% RSLogix 500 project ISO_WEEK_OF_YEAR.RSS, saved by version 9.05.01.00 %
PROJECT "ML1400"    % processor: MicroLogix 1400; MAIN_PROG %

PROGRAM FILES
  LAD 2 "MAIN_PROG"  82 rungs

DATA FILES
  O0 OUTPUT  6 elements
  I1 INPUT  8 elements
  S2 STATUS  66 elements
  B3 BINARY  53 elements
  T4 TIMER  1 elements
  C5 COUNTER  1 elements
  R6 CONTROL  1 elements
  N7 INTEGER  180 elements
  F8   1 elements

LADDER 2 "MAIN_PROG"
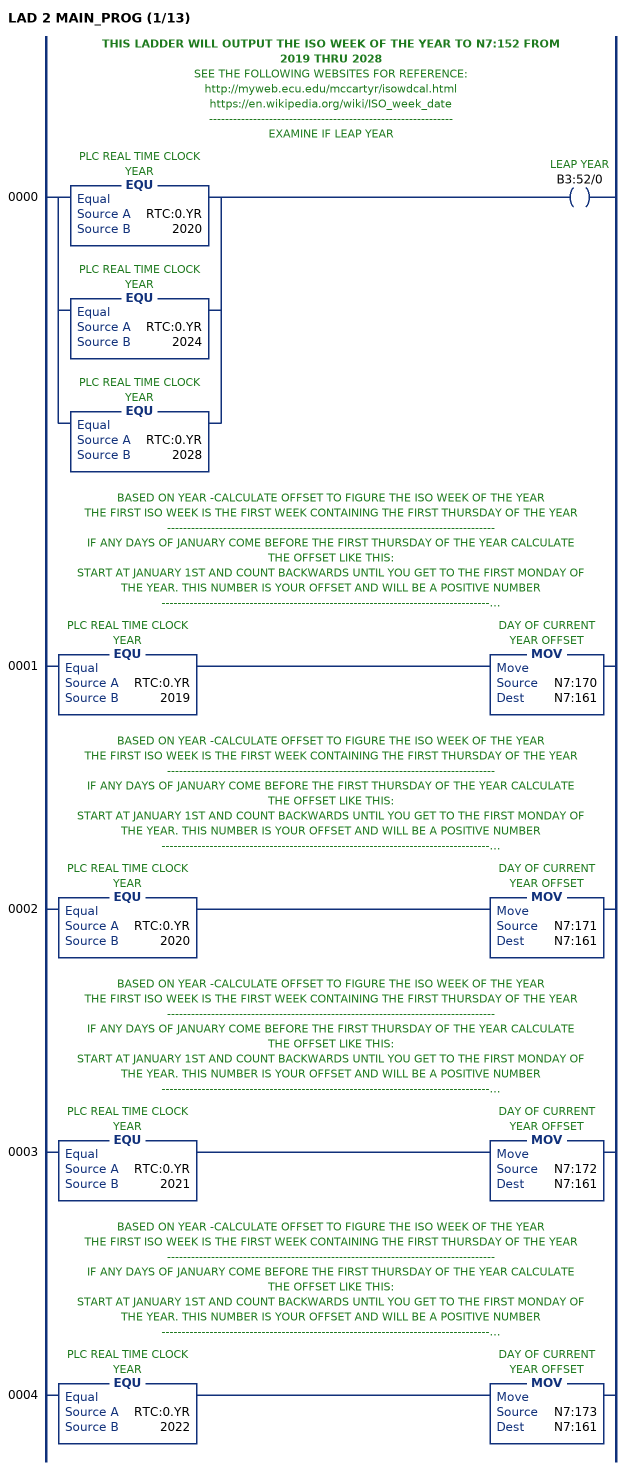
% Rung: 0 %
% TITLE: THIS LADDER WILL OUTPUT THE ISO WEEK OF THE YEAR TO N7:152 FROM 2019 THRU 2028 %
% SEE THE FOLLOWING WEBSITES FOR REFERENCE:
% http://myweb.ecu.edu/mccartyr/isowdcal.html
% https://en.wikipedia.org/wiki/ISO_week_date
% -------------------------------------------------------------
% EXAMINE IF LEAP YEAR %
SOR BST EQU RTC:0.YR 2020 NXB EQU RTC:0.YR 2024 NXB EQU RTC:0.YR 2028 BND OTE B3:52/0 EOR
%   RTC:0.YR  "PLC REAL TIME CLOCK YEAR" %
%   B3:52/0  "LEAP YEAR" %
% Rung: 1 %
% BASED ON YEAR -CALCULATE OFFSET TO FIGURE THE ISO WEEK OF THE YEAR
% THE FIRST ISO WEEK IS THE FIRST WEEK CONTAINING THE FIRST THURSDAY OF THE YEAR
% ----------------------------------------------------------------------------------
% IF ANY DAYS OF JANUARY COME BEFORE THE FIRST THURSDAY OF THE YEAR CALCULATE THE OFFSET LIKE THIS:
% START AT JANUARY 1ST AND COUNT BACKWARDS UNTIL YOU GET TO THE FIRST MONDAY OF THE YEAR. THIS NUMBER IS YOUR OFFSET AND WILL BE A POSITIVE NUMBER
% -----------------------------------------------------------------------------------
% IF NO DAYS OF JANUARY COME BEFORE THE FIRST THURSDAY OF THE YEAR CALCULATE THE OFFSET LIKE THIS:
% START AT JANUARY 1ST AND COUNT FORWARDS UNTIL YOU GET TO THE NEXT SUNDAY. THIS NUMBER IS YOUR OFFSET AND WILL BE A NEGATIVE NUMBER
% ------------------------------------------------------------------------------------
% SEE THE FOLLOWING WEBSITES FOR REFERENCE:
% http://myweb.ecu.edu/mccartyr/isowdcal.html
% https://en.wikipedia.org/wiki/ISO_week_date %
SOR EQU RTC:0.YR 2019 MOV N7:170 N7:161 EOR
%   RTC:0.YR  "PLC REAL TIME CLOCK YEAR" %
%   N7:170  "DAY OFFSET 2019" %
%   N7:161  "DAY OF CURRENT YEAR OFFSET" %
% Rung: 2 %
% BASED ON YEAR -CALCULATE OFFSET TO FIGURE THE ISO WEEK OF THE YEAR
% THE FIRST ISO WEEK IS THE FIRST WEEK CONTAINING THE FIRST THURSDAY OF THE YEAR
% ----------------------------------------------------------------------------------
% IF ANY DAYS OF JANUARY COME BEFORE THE FIRST THURSDAY OF THE YEAR CALCULATE THE OFFSET LIKE THIS:
% START AT JANUARY 1ST AND COUNT BACKWARDS UNTIL YOU GET TO THE FIRST MONDAY OF THE YEAR. THIS NUMBER IS YOUR OFFSET AND WILL BE A POSITIVE NUMBER
% -----------------------------------------------------------------------------------
% IF NO DAYS OF JANUARY COME BEFORE THE FIRST THURSDAY OF THE YEAR CALCULATE THE OFFSET LIKE THIS:
% START AT JANUARY 1ST AND COUNT FORWARDS UNTIL YOU GET TO THE NEXT SUNDAY. THIS NUMBER IS YOUR OFFSET AND WILL BE A NEGATIVE NUMBER
% ------------------------------------------------------------------------------------
% SEE THE FOLLOWING WEBSITES FOR REFERENCE:
% http://myweb.ecu.edu/mccartyr/isowdcal.html
% https://en.wikipedia.org/wiki/ISO_week_date %
SOR EQU RTC:0.YR 2020 MOV N7:171 N7:161 EOR
%   RTC:0.YR  "PLC REAL TIME CLOCK YEAR" %
%   N7:171  "DAY OFFSET 2020" %
%   N7:161  "DAY OF CURRENT YEAR OFFSET" %
% Rung: 3 %
% BASED ON YEAR -CALCULATE OFFSET TO FIGURE THE ISO WEEK OF THE YEAR
% THE FIRST ISO WEEK IS THE FIRST WEEK CONTAINING THE FIRST THURSDAY OF THE YEAR
% ----------------------------------------------------------------------------------
% IF ANY DAYS OF JANUARY COME BEFORE THE FIRST THURSDAY OF THE YEAR CALCULATE THE OFFSET LIKE THIS:
% START AT JANUARY 1ST AND COUNT BACKWARDS UNTIL YOU GET TO THE FIRST MONDAY OF THE YEAR. THIS NUMBER IS YOUR OFFSET AND WILL BE A POSITIVE NUMBER
% -----------------------------------------------------------------------------------
% IF NO DAYS OF JANUARY COME BEFORE THE FIRST THURSDAY OF THE YEAR CALCULATE THE OFFSET LIKE THIS:
% START AT JANUARY 1ST AND COUNT FORWARDS UNTIL YOU GET TO THE NEXT SUNDAY. THIS NUMBER IS YOUR OFFSET AND WILL BE A NEGATIVE NUMBER
% ------------------------------------------------------------------------------------
% SEE THE FOLLOWING WEBSITES FOR REFERENCE:
% http://myweb.ecu.edu/mccartyr/isowdcal.html
% https://en.wikipedia.org/wiki/ISO_week_date %
SOR EQU RTC:0.YR 2021 MOV N7:172 N7:161 EOR
%   RTC:0.YR  "PLC REAL TIME CLOCK YEAR" %
%   N7:172  "DAY OFFSET 2021" %
%   N7:161  "DAY OF CURRENT YEAR OFFSET" %
% Rung: 4 %
% BASED ON YEAR -CALCULATE OFFSET TO FIGURE THE ISO WEEK OF THE YEAR
% THE FIRST ISO WEEK IS THE FIRST WEEK CONTAINING THE FIRST THURSDAY OF THE YEAR
% ----------------------------------------------------------------------------------
% IF ANY DAYS OF JANUARY COME BEFORE THE FIRST THURSDAY OF THE YEAR CALCULATE THE OFFSET LIKE THIS:
% START AT JANUARY 1ST AND COUNT BACKWARDS UNTIL YOU GET TO THE FIRST MONDAY OF THE YEAR. THIS NUMBER IS YOUR OFFSET AND WILL BE A POSITIVE NUMBER
% -----------------------------------------------------------------------------------
% IF NO DAYS OF JANUARY COME BEFORE THE FIRST THURSDAY OF THE YEAR CALCULATE THE OFFSET LIKE THIS:
% START AT JANUARY 1ST AND COUNT FORWARDS UNTIL YOU GET TO THE NEXT SUNDAY. THIS NUMBER IS YOUR OFFSET AND WILL BE A NEGATIVE NUMBER
% ------------------------------------------------------------------------------------
% SEE THE FOLLOWING WEBSITES FOR REFERENCE:
% http://myweb.ecu.edu/mccartyr/isowdcal.html
% https://en.wikipedia.org/wiki/ISO_week_date %
SOR EQU RTC:0.YR 2022 MOV N7:173 N7:161 EOR
%   RTC:0.YR  "PLC REAL TIME CLOCK YEAR" %
%   N7:173  "DAY OFFSET 2022" %
%   N7:161  "DAY OF CURRENT YEAR OFFSET" %

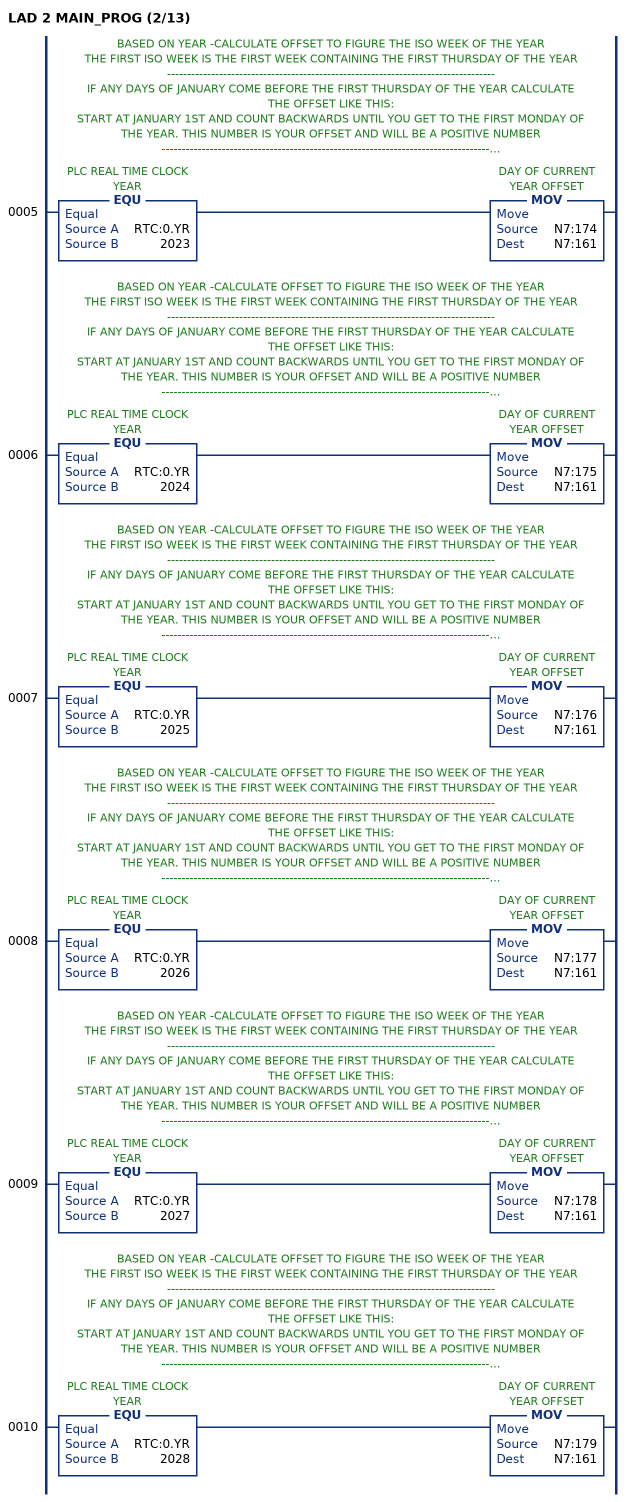
% Rung: 5 %
% BASED ON YEAR -CALCULATE OFFSET TO FIGURE THE ISO WEEK OF THE YEAR
% THE FIRST ISO WEEK IS THE FIRST WEEK CONTAINING THE FIRST THURSDAY OF THE YEAR
% ----------------------------------------------------------------------------------
% IF ANY DAYS OF JANUARY COME BEFORE THE FIRST THURSDAY OF THE YEAR CALCULATE THE OFFSET LIKE THIS:
% START AT JANUARY 1ST AND COUNT BACKWARDS UNTIL YOU GET TO THE FIRST MONDAY OF THE YEAR. THIS NUMBER IS YOUR OFFSET AND WILL BE A POSITIVE NUMBER
% -----------------------------------------------------------------------------------
% IF NO DAYS OF JANUARY COME BEFORE THE FIRST THURSDAY OF THE YEAR CALCULATE THE OFFSET LIKE THIS:
% START AT JANUARY 1ST AND COUNT FORWARDS UNTIL YOU GET TO THE NEXT SUNDAY. THIS NUMBER IS YOUR OFFSET AND WILL BE A NEGATIVE NUMBER
% ------------------------------------------------------------------------------------
% SEE THE FOLLOWING WEBSITES FOR REFERENCE:
% http://myweb.ecu.edu/mccartyr/isowdcal.html
% https://en.wikipedia.org/wiki/ISO_week_date %
SOR EQU RTC:0.YR 2023 MOV N7:174 N7:161 EOR
%   RTC:0.YR  "PLC REAL TIME CLOCK YEAR" %
%   N7:174  "DAY OFFSET 2023" %
%   N7:161  "DAY OF CURRENT YEAR OFFSET" %
% Rung: 6 %
% BASED ON YEAR -CALCULATE OFFSET TO FIGURE THE ISO WEEK OF THE YEAR
% THE FIRST ISO WEEK IS THE FIRST WEEK CONTAINING THE FIRST THURSDAY OF THE YEAR
% ----------------------------------------------------------------------------------
% IF ANY DAYS OF JANUARY COME BEFORE THE FIRST THURSDAY OF THE YEAR CALCULATE THE OFFSET LIKE THIS:
% START AT JANUARY 1ST AND COUNT BACKWARDS UNTIL YOU GET TO THE FIRST MONDAY OF THE YEAR. THIS NUMBER IS YOUR OFFSET AND WILL BE A POSITIVE NUMBER
% -----------------------------------------------------------------------------------
% IF NO DAYS OF JANUARY COME BEFORE THE FIRST THURSDAY OF THE YEAR CALCULATE THE OFFSET LIKE THIS:
% START AT JANUARY 1ST AND COUNT FORWARDS UNTIL YOU GET TO THE NEXT SUNDAY. THIS NUMBER IS YOUR OFFSET AND WILL BE A NEGATIVE NUMBER
% ------------------------------------------------------------------------------------
% SEE THE FOLLOWING WEBSITES FOR REFERENCE:
% http://myweb.ecu.edu/mccartyr/isowdcal.html
% https://en.wikipedia.org/wiki/ISO_week_date %
SOR EQU RTC:0.YR 2024 MOV N7:175 N7:161 EOR
%   RTC:0.YR  "PLC REAL TIME CLOCK YEAR" %
%   N7:175  "DAY OFFSET 2024" %
%   N7:161  "DAY OF CURRENT YEAR OFFSET" %
% Rung: 7 %
% BASED ON YEAR -CALCULATE OFFSET TO FIGURE THE ISO WEEK OF THE YEAR
% THE FIRST ISO WEEK IS THE FIRST WEEK CONTAINING THE FIRST THURSDAY OF THE YEAR
% ----------------------------------------------------------------------------------
% IF ANY DAYS OF JANUARY COME BEFORE THE FIRST THURSDAY OF THE YEAR CALCULATE THE OFFSET LIKE THIS:
% START AT JANUARY 1ST AND COUNT BACKWARDS UNTIL YOU GET TO THE FIRST MONDAY OF THE YEAR. THIS NUMBER IS YOUR OFFSET AND WILL BE A POSITIVE NUMBER
% -----------------------------------------------------------------------------------
% IF NO DAYS OF JANUARY COME BEFORE THE FIRST THURSDAY OF THE YEAR CALCULATE THE OFFSET LIKE THIS:
% START AT JANUARY 1ST AND COUNT FORWARDS UNTIL YOU GET TO THE NEXT SUNDAY. THIS NUMBER IS YOUR OFFSET AND WILL BE A NEGATIVE NUMBER
% ------------------------------------------------------------------------------------
% SEE THE FOLLOWING WEBSITES FOR REFERENCE:
% http://myweb.ecu.edu/mccartyr/isowdcal.html
% https://en.wikipedia.org/wiki/ISO_week_date %
SOR EQU RTC:0.YR 2025 MOV N7:176 N7:161 EOR
%   RTC:0.YR  "PLC REAL TIME CLOCK YEAR" %
%   N7:176  "DAY OFFSET 2025" %
%   N7:161  "DAY OF CURRENT YEAR OFFSET" %
% Rung: 8 %
% BASED ON YEAR -CALCULATE OFFSET TO FIGURE THE ISO WEEK OF THE YEAR
% THE FIRST ISO WEEK IS THE FIRST WEEK CONTAINING THE FIRST THURSDAY OF THE YEAR
% ----------------------------------------------------------------------------------
% IF ANY DAYS OF JANUARY COME BEFORE THE FIRST THURSDAY OF THE YEAR CALCULATE THE OFFSET LIKE THIS:
% START AT JANUARY 1ST AND COUNT BACKWARDS UNTIL YOU GET TO THE FIRST MONDAY OF THE YEAR. THIS NUMBER IS YOUR OFFSET AND WILL BE A POSITIVE NUMBER
% -----------------------------------------------------------------------------------
% IF NO DAYS OF JANUARY COME BEFORE THE FIRST THURSDAY OF THE YEAR CALCULATE THE OFFSET LIKE THIS:
% START AT JANUARY 1ST AND COUNT FORWARDS UNTIL YOU GET TO THE NEXT SUNDAY. THIS NUMBER IS YOUR OFFSET AND WILL BE A NEGATIVE NUMBER
% ------------------------------------------------------------------------------------
% SEE THE FOLLOWING WEBSITES FOR REFERENCE:
% http://myweb.ecu.edu/mccartyr/isowdcal.html
% https://en.wikipedia.org/wiki/ISO_week_date %
SOR EQU RTC:0.YR 2026 MOV N7:177 N7:161 EOR
%   RTC:0.YR  "PLC REAL TIME CLOCK YEAR" %
%   N7:177  "DAY OFFSET 2026" %
%   N7:161  "DAY OF CURRENT YEAR OFFSET" %
% Rung: 9 %
% BASED ON YEAR -CALCULATE OFFSET TO FIGURE THE ISO WEEK OF THE YEAR
% THE FIRST ISO WEEK IS THE FIRST WEEK CONTAINING THE FIRST THURSDAY OF THE YEAR
% ----------------------------------------------------------------------------------
% IF ANY DAYS OF JANUARY COME BEFORE THE FIRST THURSDAY OF THE YEAR CALCULATE THE OFFSET LIKE THIS:
% START AT JANUARY 1ST AND COUNT BACKWARDS UNTIL YOU GET TO THE FIRST MONDAY OF THE YEAR. THIS NUMBER IS YOUR OFFSET AND WILL BE A POSITIVE NUMBER
% -----------------------------------------------------------------------------------
% IF NO DAYS OF JANUARY COME BEFORE THE FIRST THURSDAY OF THE YEAR CALCULATE THE OFFSET LIKE THIS:
% START AT JANUARY 1ST AND COUNT FORWARDS UNTIL YOU GET TO THE NEXT SUNDAY. THIS NUMBER IS YOUR OFFSET AND WILL BE A NEGATIVE NUMBER
% ------------------------------------------------------------------------------------
% SEE THE FOLLOWING WEBSITES FOR REFERENCE:
% http://myweb.ecu.edu/mccartyr/isowdcal.html
% https://en.wikipedia.org/wiki/ISO_week_date %
SOR EQU RTC:0.YR 2027 MOV N7:178 N7:161 EOR
%   RTC:0.YR  "PLC REAL TIME CLOCK YEAR" %
%   N7:178  "DAY OFFSET 2027" %
%   N7:161  "DAY OF CURRENT YEAR OFFSET" %
% Rung: 10 %
% BASED ON YEAR -CALCULATE OFFSET TO FIGURE THE ISO WEEK OF THE YEAR
% THE FIRST ISO WEEK IS THE FIRST WEEK CONTAINING THE FIRST THURSDAY OF THE YEAR
% ----------------------------------------------------------------------------------
% IF ANY DAYS OF JANUARY COME BEFORE THE FIRST THURSDAY OF THE YEAR CALCULATE THE OFFSET LIKE THIS:
% START AT JANUARY 1ST AND COUNT BACKWARDS UNTIL YOU GET TO THE FIRST MONDAY OF THE YEAR. THIS NUMBER IS YOUR OFFSET AND WILL BE A POSITIVE NUMBER
% -----------------------------------------------------------------------------------
% IF NO DAYS OF JANUARY COME BEFORE THE FIRST THURSDAY OF THE YEAR CALCULATE THE OFFSET LIKE THIS:
% START AT JANUARY 1ST AND COUNT FORWARDS UNTIL YOU GET TO THE NEXT SUNDAY. THIS NUMBER IS YOUR OFFSET AND WILL BE A NEGATIVE NUMBER
% ------------------------------------------------------------------------------------
% SEE THE FOLLOWING WEBSITES FOR REFERENCE:
% http://myweb.ecu.edu/mccartyr/isowdcal.html
% https://en.wikipedia.org/wiki/ISO_week_date %
SOR EQU RTC:0.YR 2028 MOV N7:179 N7:161 EOR
%   RTC:0.YR  "PLC REAL TIME CLOCK YEAR" %
%   N7:179  "DAY OFFSET 2028" %
%   N7:161  "DAY OF CURRENT YEAR OFFSET" %

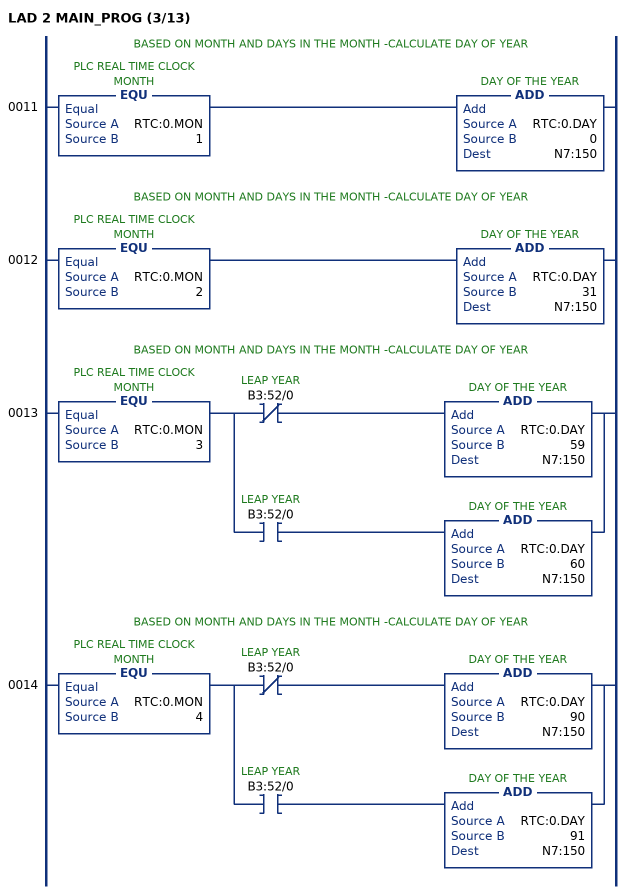
% Rung: 11 %
% BASED ON MONTH AND DAYS IN THE MONTH -CALCULATE DAY OF YEAR %
SOR EQU RTC:0.MON 1 ADD RTC:0.DAY 0 N7:150 EOR
%   RTC:0.MON  "PLC REAL TIME CLOCK MONTH" %
%   RTC:0.DAY  "PLC REAL TIME CLOCK DAY" %
%   N7:150  "DAY OF THE YEAR" %
% Rung: 12 %
% BASED ON MONTH AND DAYS IN THE MONTH -CALCULATE DAY OF YEAR %
SOR EQU RTC:0.MON 2 ADD RTC:0.DAY 31 N7:150 EOR
%   RTC:0.MON  "PLC REAL TIME CLOCK MONTH" %
%   RTC:0.DAY  "PLC REAL TIME CLOCK DAY" %
%   N7:150  "DAY OF THE YEAR" %
% Rung: 13 %
% BASED ON MONTH AND DAYS IN THE MONTH -CALCULATE DAY OF YEAR %
SOR EQU RTC:0.MON 3 BST XIO B3:52/0 ADD RTC:0.DAY 59 N7:150 NXB XIC B3:52/0 ADD RTC:0.DAY 60 N7:150 BND EOR
%   RTC:0.MON  "PLC REAL TIME CLOCK MONTH" %
%   B3:52/0  "LEAP YEAR" %
%   RTC:0.DAY  "PLC REAL TIME CLOCK DAY" %
%   N7:150  "DAY OF THE YEAR" %
% Rung: 14 %
% BASED ON MONTH AND DAYS IN THE MONTH -CALCULATE DAY OF YEAR %
SOR EQU RTC:0.MON 4 BST XIO B3:52/0 ADD RTC:0.DAY 90 N7:150 NXB XIC B3:52/0 ADD RTC:0.DAY 91 N7:150 BND EOR
%   RTC:0.MON  "PLC REAL TIME CLOCK MONTH" %
%   B3:52/0  "LEAP YEAR" %
%   RTC:0.DAY  "PLC REAL TIME CLOCK DAY" %
%   N7:150  "DAY OF THE YEAR" %

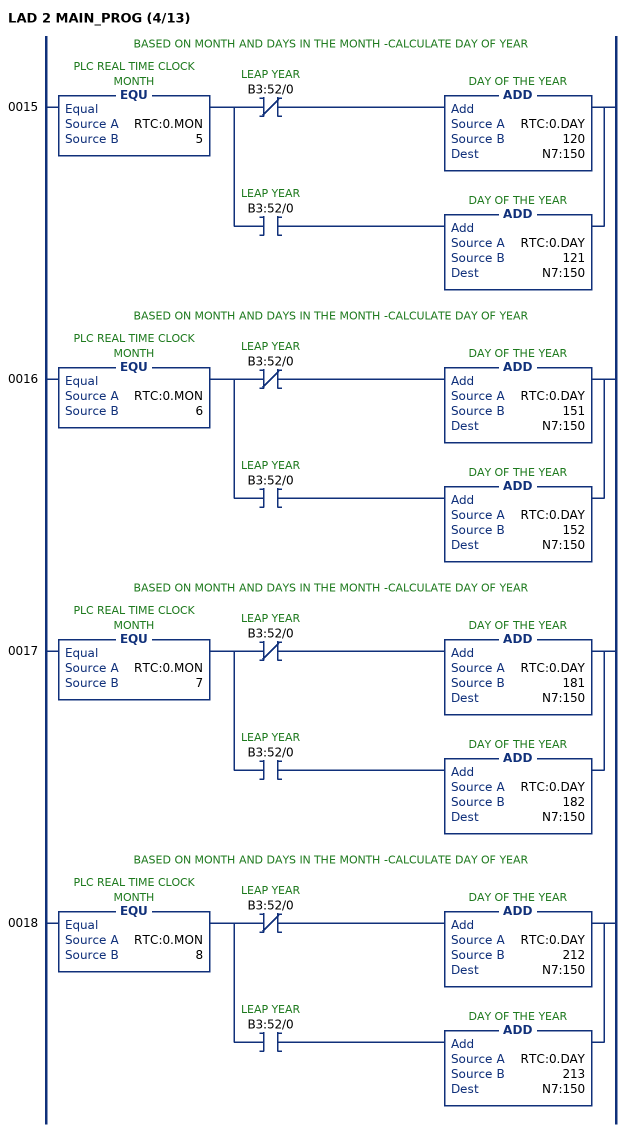
% Rung: 15 %
% BASED ON MONTH AND DAYS IN THE MONTH -CALCULATE DAY OF YEAR %
SOR EQU RTC:0.MON 5 BST XIO B3:52/0 ADD RTC:0.DAY 120 N7:150 NXB XIC B3:52/0 ADD RTC:0.DAY 121 N7:150 BND EOR
%   RTC:0.MON  "PLC REAL TIME CLOCK MONTH" %
%   B3:52/0  "LEAP YEAR" %
%   RTC:0.DAY  "PLC REAL TIME CLOCK DAY" %
%   N7:150  "DAY OF THE YEAR" %
% Rung: 16 %
% BASED ON MONTH AND DAYS IN THE MONTH -CALCULATE DAY OF YEAR %
SOR EQU RTC:0.MON 6 BST XIO B3:52/0 ADD RTC:0.DAY 151 N7:150 NXB XIC B3:52/0 ADD RTC:0.DAY 152 N7:150 BND EOR
%   RTC:0.MON  "PLC REAL TIME CLOCK MONTH" %
%   B3:52/0  "LEAP YEAR" %
%   RTC:0.DAY  "PLC REAL TIME CLOCK DAY" %
%   N7:150  "DAY OF THE YEAR" %
% Rung: 17 %
% BASED ON MONTH AND DAYS IN THE MONTH -CALCULATE DAY OF YEAR %
SOR EQU RTC:0.MON 7 BST XIO B3:52/0 ADD RTC:0.DAY 181 N7:150 NXB XIC B3:52/0 ADD RTC:0.DAY 182 N7:150 BND EOR
%   RTC:0.MON  "PLC REAL TIME CLOCK MONTH" %
%   B3:52/0  "LEAP YEAR" %
%   RTC:0.DAY  "PLC REAL TIME CLOCK DAY" %
%   N7:150  "DAY OF THE YEAR" %
% Rung: 18 %
% BASED ON MONTH AND DAYS IN THE MONTH -CALCULATE DAY OF YEAR %
SOR EQU RTC:0.MON 8 BST XIO B3:52/0 ADD RTC:0.DAY 212 N7:150 NXB XIC B3:52/0 ADD RTC:0.DAY 213 N7:150 BND EOR
%   RTC:0.MON  "PLC REAL TIME CLOCK MONTH" %
%   B3:52/0  "LEAP YEAR" %
%   RTC:0.DAY  "PLC REAL TIME CLOCK DAY" %
%   N7:150  "DAY OF THE YEAR" %

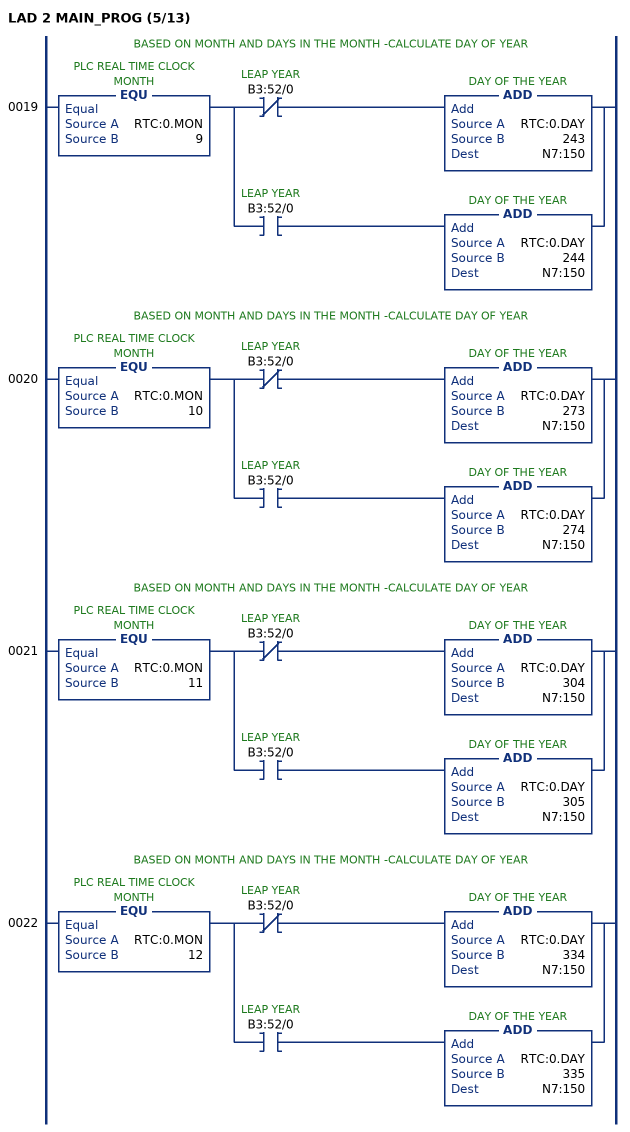
% Rung: 19 %
% BASED ON MONTH AND DAYS IN THE MONTH -CALCULATE DAY OF YEAR %
SOR EQU RTC:0.MON 9 BST XIO B3:52/0 ADD RTC:0.DAY 243 N7:150 NXB XIC B3:52/0 ADD RTC:0.DAY 244 N7:150 BND EOR
%   RTC:0.MON  "PLC REAL TIME CLOCK MONTH" %
%   B3:52/0  "LEAP YEAR" %
%   RTC:0.DAY  "PLC REAL TIME CLOCK DAY" %
%   N7:150  "DAY OF THE YEAR" %
% Rung: 20 %
% BASED ON MONTH AND DAYS IN THE MONTH -CALCULATE DAY OF YEAR %
SOR EQU RTC:0.MON 10 BST XIO B3:52/0 ADD RTC:0.DAY 273 N7:150 NXB XIC B3:52/0 ADD RTC:0.DAY 274 N7:150 BND EOR
%   RTC:0.MON  "PLC REAL TIME CLOCK MONTH" %
%   B3:52/0  "LEAP YEAR" %
%   RTC:0.DAY  "PLC REAL TIME CLOCK DAY" %
%   N7:150  "DAY OF THE YEAR" %
% Rung: 21 %
% BASED ON MONTH AND DAYS IN THE MONTH -CALCULATE DAY OF YEAR %
SOR EQU RTC:0.MON 11 BST XIO B3:52/0 ADD RTC:0.DAY 304 N7:150 NXB XIC B3:52/0 ADD RTC:0.DAY 305 N7:150 BND EOR
%   RTC:0.MON  "PLC REAL TIME CLOCK MONTH" %
%   B3:52/0  "LEAP YEAR" %
%   RTC:0.DAY  "PLC REAL TIME CLOCK DAY" %
%   N7:150  "DAY OF THE YEAR" %
% Rung: 22 %
% BASED ON MONTH AND DAYS IN THE MONTH -CALCULATE DAY OF YEAR %
SOR EQU RTC:0.MON 12 BST XIO B3:52/0 ADD RTC:0.DAY 334 N7:150 NXB XIC B3:52/0 ADD RTC:0.DAY 335 N7:150 BND EOR
%   RTC:0.MON  "PLC REAL TIME CLOCK MONTH" %
%   B3:52/0  "LEAP YEAR" %
%   RTC:0.DAY  "PLC REAL TIME CLOCK DAY" %
%   N7:150  "DAY OF THE YEAR" %

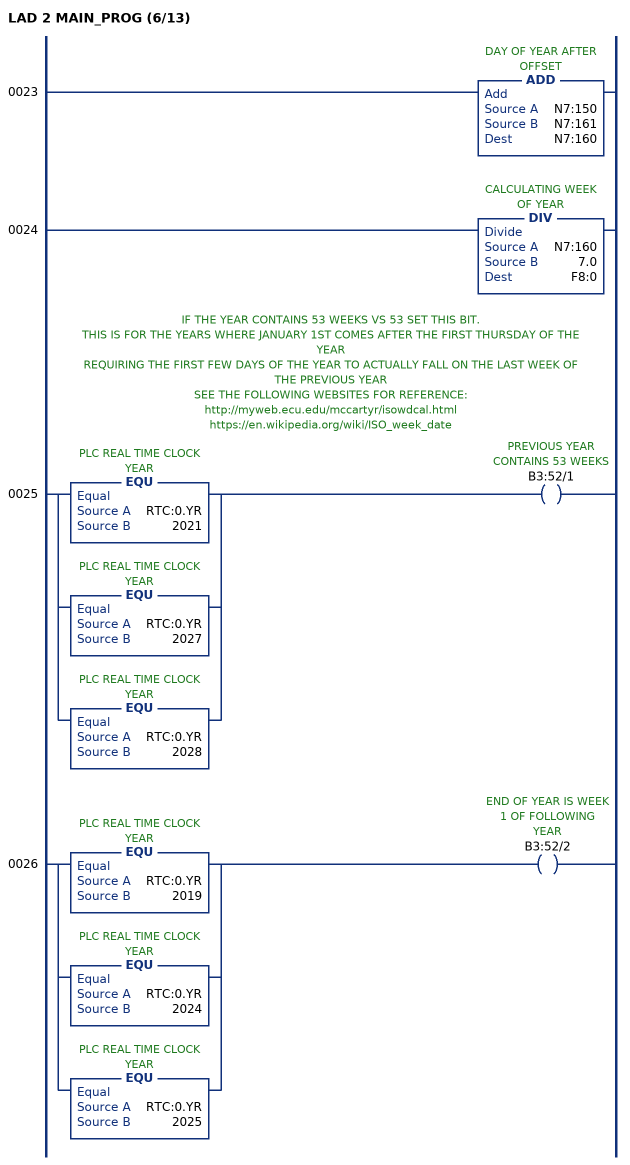
% Rung: 23 %
SOR ADD N7:150 N7:161 N7:160 EOR
%   N7:150  "DAY OF THE YEAR" %
%   N7:161  "DAY OF CURRENT YEAR OFFSET" %
%   N7:160  "DAY OF YEAR AFTER OFFSET" %
% Rung: 24 %
SOR DIV N7:160 7.0 F8:0 EOR
%   N7:160  "DAY OF YEAR AFTER OFFSET" %
%   F8:0  "CALCULATING WEEK OF YEAR" %
% Rung: 25 %
% IF THE YEAR CONTAINS 53 WEEKS VS 53 SET THIS BIT.
% THIS IS FOR THE YEARS WHERE JANUARY 1ST COMES AFTER THE FIRST THURSDAY OF THE YEAR
% REQUIRING THE FIRST FEW DAYS OF THE YEAR TO ACTUALLY FALL ON THE LAST WEEK OF THE PREVIOUS YEAR
% SEE THE FOLLOWING WEBSITES FOR REFERENCE:
% http://myweb.ecu.edu/mccartyr/isowdcal.html
% https://en.wikipedia.org/wiki/ISO_week_date %
SOR BST EQU RTC:0.YR 2021 NXB EQU RTC:0.YR 2027 NXB EQU RTC:0.YR 2028 BND OTE B3:52/1 EOR
%   RTC:0.YR  "PLC REAL TIME CLOCK YEAR" %
%   B3:52/1  "PREVIOUS YEAR CONTAINS 53 WEEKS" %
% Rung: 26 %
SOR BST EQU RTC:0.YR 2019 NXB EQU RTC:0.YR 2024 NXB EQU RTC:0.YR 2025 BND OTE B3:52/2 EOR
%   RTC:0.YR  "PLC REAL TIME CLOCK YEAR" %
%   B3:52/2  "END OF YEAR IS WEEK 1 OF FOLLOWING YEAR" %

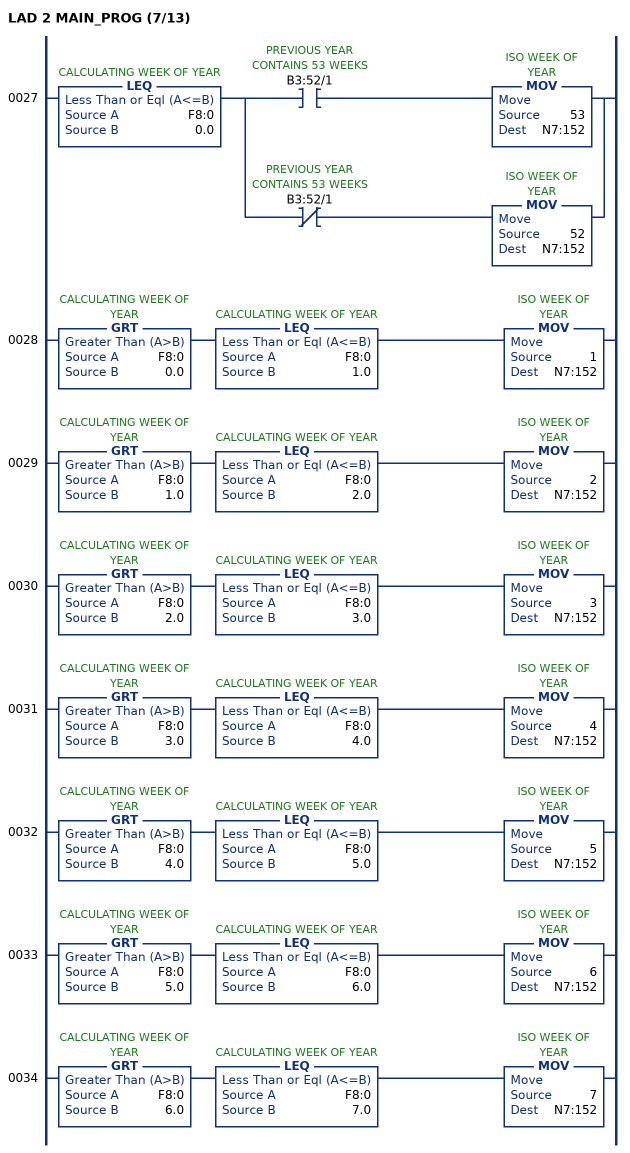
% Rung: 27 %
SOR LEQ F8:0 0.0 BST XIC B3:52/1 MOV 53 N7:152 NXB XIO B3:52/1 MOV 52 N7:152 BND EOR
%   F8:0  "CALCULATING WEEK OF YEAR" %
%   B3:52/1  "PREVIOUS YEAR CONTAINS 53 WEEKS" %
%   N7:152  "ISO WEEK OF YEAR" %
% Rung: 28 %
SOR GRT F8:0 0.0 LEQ F8:0 1.0 MOV 1 N7:152 EOR
%   F8:0  "CALCULATING WEEK OF YEAR" %
%   N7:152  "ISO WEEK OF YEAR" %
% Rung: 29 %
SOR GRT F8:0 1.0 LEQ F8:0 2.0 MOV 2 N7:152 EOR
%   F8:0  "CALCULATING WEEK OF YEAR" %
%   N7:152  "ISO WEEK OF YEAR" %
% Rung: 30 %
SOR GRT F8:0 2.0 LEQ F8:0 3.0 MOV 3 N7:152 EOR
%   F8:0  "CALCULATING WEEK OF YEAR" %
%   N7:152  "ISO WEEK OF YEAR" %
% Rung: 31 %
SOR GRT F8:0 3.0 LEQ F8:0 4.0 MOV 4 N7:152 EOR
%   F8:0  "CALCULATING WEEK OF YEAR" %
%   N7:152  "ISO WEEK OF YEAR" %
% Rung: 32 %
SOR GRT F8:0 4.0 LEQ F8:0 5.0 MOV 5 N7:152 EOR
%   F8:0  "CALCULATING WEEK OF YEAR" %
%   N7:152  "ISO WEEK OF YEAR" %
% Rung: 33 %
SOR GRT F8:0 5.0 LEQ F8:0 6.0 MOV 6 N7:152 EOR
%   F8:0  "CALCULATING WEEK OF YEAR" %
%   N7:152  "ISO WEEK OF YEAR" %
% Rung: 34 %
SOR GRT F8:0 6.0 LEQ F8:0 7.0 MOV 7 N7:152 EOR
%   F8:0  "CALCULATING WEEK OF YEAR" %
%   N7:152  "ISO WEEK OF YEAR" %

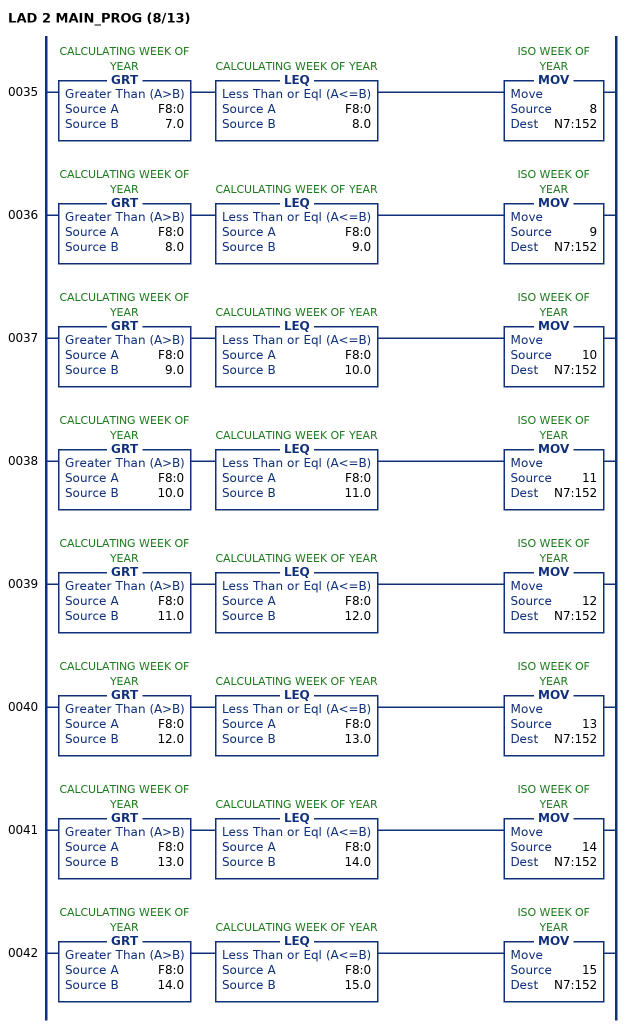
% Rung: 35 %
SOR GRT F8:0 7.0 LEQ F8:0 8.0 MOV 8 N7:152 EOR
%   F8:0  "CALCULATING WEEK OF YEAR" %
%   N7:152  "ISO WEEK OF YEAR" %
% Rung: 36 %
SOR GRT F8:0 8.0 LEQ F8:0 9.0 MOV 9 N7:152 EOR
%   F8:0  "CALCULATING WEEK OF YEAR" %
%   N7:152  "ISO WEEK OF YEAR" %
% Rung: 37 %
SOR GRT F8:0 9.0 LEQ F8:0 10.0 MOV 10 N7:152 EOR
%   F8:0  "CALCULATING WEEK OF YEAR" %
%   N7:152  "ISO WEEK OF YEAR" %
% Rung: 38 %
SOR GRT F8:0 10.0 LEQ F8:0 11.0 MOV 11 N7:152 EOR
%   F8:0  "CALCULATING WEEK OF YEAR" %
%   N7:152  "ISO WEEK OF YEAR" %
% Rung: 39 %
SOR GRT F8:0 11.0 LEQ F8:0 12.0 MOV 12 N7:152 EOR
%   F8:0  "CALCULATING WEEK OF YEAR" %
%   N7:152  "ISO WEEK OF YEAR" %
% Rung: 40 %
SOR GRT F8:0 12.0 LEQ F8:0 13.0 MOV 13 N7:152 EOR
%   F8:0  "CALCULATING WEEK OF YEAR" %
%   N7:152  "ISO WEEK OF YEAR" %
% Rung: 41 %
SOR GRT F8:0 13.0 LEQ F8:0 14.0 MOV 14 N7:152 EOR
%   F8:0  "CALCULATING WEEK OF YEAR" %
%   N7:152  "ISO WEEK OF YEAR" %
% Rung: 42 %
SOR GRT F8:0 14.0 LEQ F8:0 15.0 MOV 15 N7:152 EOR
%   F8:0  "CALCULATING WEEK OF YEAR" %
%   N7:152  "ISO WEEK OF YEAR" %

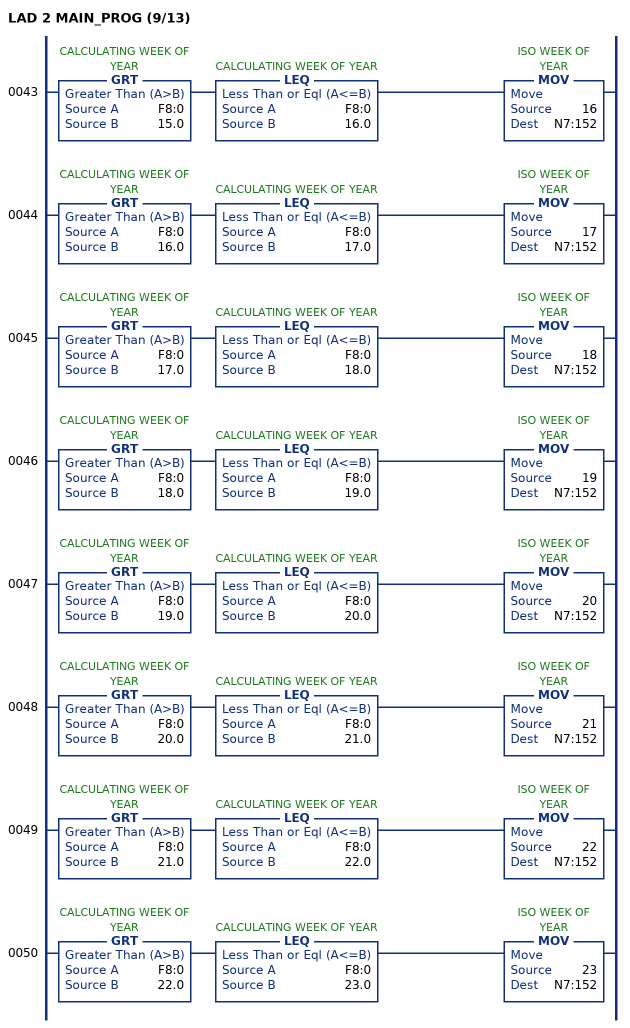
% Rung: 43 %
SOR GRT F8:0 15.0 LEQ F8:0 16.0 MOV 16 N7:152 EOR
%   F8:0  "CALCULATING WEEK OF YEAR" %
%   N7:152  "ISO WEEK OF YEAR" %
% Rung: 44 %
SOR GRT F8:0 16.0 LEQ F8:0 17.0 MOV 17 N7:152 EOR
%   F8:0  "CALCULATING WEEK OF YEAR" %
%   N7:152  "ISO WEEK OF YEAR" %
% Rung: 45 %
SOR GRT F8:0 17.0 LEQ F8:0 18.0 MOV 18 N7:152 EOR
%   F8:0  "CALCULATING WEEK OF YEAR" %
%   N7:152  "ISO WEEK OF YEAR" %
% Rung: 46 %
SOR GRT F8:0 18.0 LEQ F8:0 19.0 MOV 19 N7:152 EOR
%   F8:0  "CALCULATING WEEK OF YEAR" %
%   N7:152  "ISO WEEK OF YEAR" %
% Rung: 47 %
SOR GRT F8:0 19.0 LEQ F8:0 20.0 MOV 20 N7:152 EOR
%   F8:0  "CALCULATING WEEK OF YEAR" %
%   N7:152  "ISO WEEK OF YEAR" %
% Rung: 48 %
SOR GRT F8:0 20.0 LEQ F8:0 21.0 MOV 21 N7:152 EOR
%   F8:0  "CALCULATING WEEK OF YEAR" %
%   N7:152  "ISO WEEK OF YEAR" %
% Rung: 49 %
SOR GRT F8:0 21.0 LEQ F8:0 22.0 MOV 22 N7:152 EOR
%   F8:0  "CALCULATING WEEK OF YEAR" %
%   N7:152  "ISO WEEK OF YEAR" %
% Rung: 50 %
SOR GRT F8:0 22.0 LEQ F8:0 23.0 MOV 23 N7:152 EOR
%   F8:0  "CALCULATING WEEK OF YEAR" %
%   N7:152  "ISO WEEK OF YEAR" %

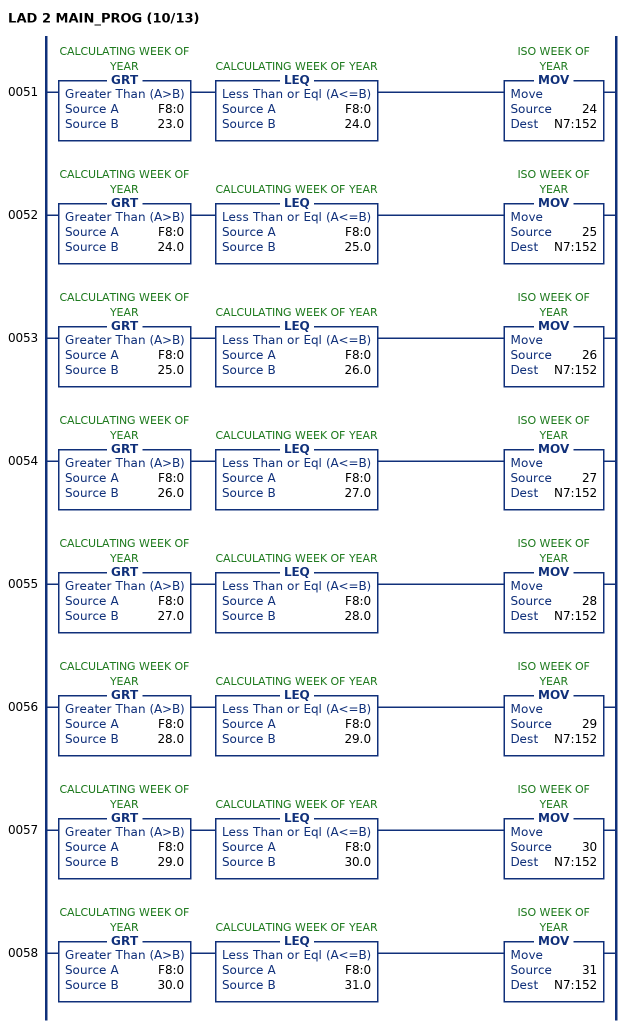
% Rung: 51 %
SOR GRT F8:0 23.0 LEQ F8:0 24.0 MOV 24 N7:152 EOR
%   F8:0  "CALCULATING WEEK OF YEAR" %
%   N7:152  "ISO WEEK OF YEAR" %
% Rung: 52 %
SOR GRT F8:0 24.0 LEQ F8:0 25.0 MOV 25 N7:152 EOR
%   F8:0  "CALCULATING WEEK OF YEAR" %
%   N7:152  "ISO WEEK OF YEAR" %
% Rung: 53 %
SOR GRT F8:0 25.0 LEQ F8:0 26.0 MOV 26 N7:152 EOR
%   F8:0  "CALCULATING WEEK OF YEAR" %
%   N7:152  "ISO WEEK OF YEAR" %
% Rung: 54 %
SOR GRT F8:0 26.0 LEQ F8:0 27.0 MOV 27 N7:152 EOR
%   F8:0  "CALCULATING WEEK OF YEAR" %
%   N7:152  "ISO WEEK OF YEAR" %
% Rung: 55 %
SOR GRT F8:0 27.0 LEQ F8:0 28.0 MOV 28 N7:152 EOR
%   F8:0  "CALCULATING WEEK OF YEAR" %
%   N7:152  "ISO WEEK OF YEAR" %
% Rung: 56 %
SOR GRT F8:0 28.0 LEQ F8:0 29.0 MOV 29 N7:152 EOR
%   F8:0  "CALCULATING WEEK OF YEAR" %
%   N7:152  "ISO WEEK OF YEAR" %
% Rung: 57 %
SOR GRT F8:0 29.0 LEQ F8:0 30.0 MOV 30 N7:152 EOR
%   F8:0  "CALCULATING WEEK OF YEAR" %
%   N7:152  "ISO WEEK OF YEAR" %
% Rung: 58 %
SOR GRT F8:0 30.0 LEQ F8:0 31.0 MOV 31 N7:152 EOR
%   F8:0  "CALCULATING WEEK OF YEAR" %
%   N7:152  "ISO WEEK OF YEAR" %

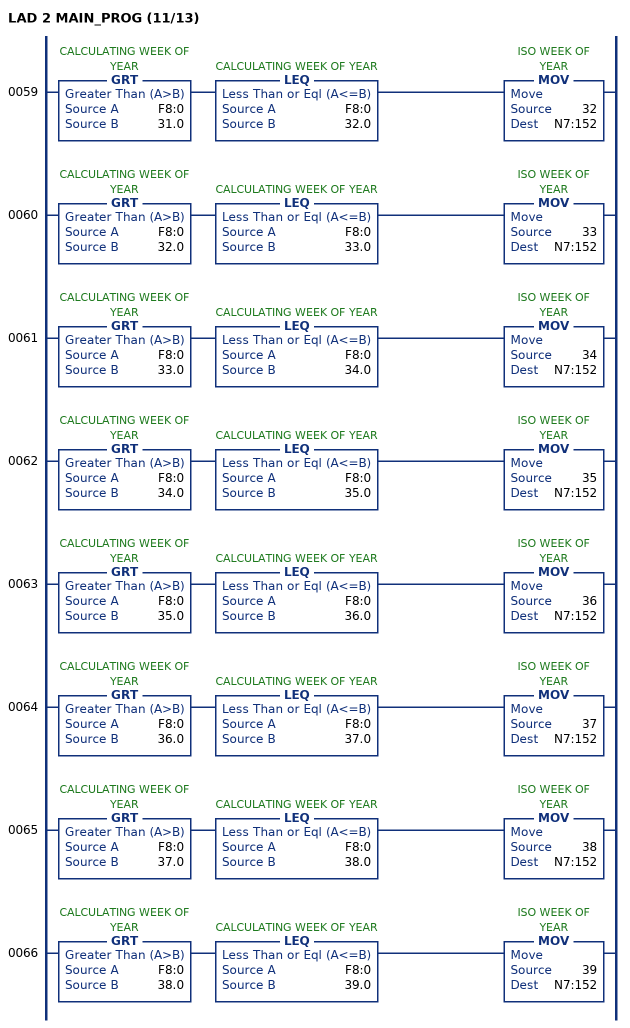
% Rung: 59 %
SOR GRT F8:0 31.0 LEQ F8:0 32.0 MOV 32 N7:152 EOR
%   F8:0  "CALCULATING WEEK OF YEAR" %
%   N7:152  "ISO WEEK OF YEAR" %
% Rung: 60 %
SOR GRT F8:0 32.0 LEQ F8:0 33.0 MOV 33 N7:152 EOR
%   F8:0  "CALCULATING WEEK OF YEAR" %
%   N7:152  "ISO WEEK OF YEAR" %
% Rung: 61 %
SOR GRT F8:0 33.0 LEQ F8:0 34.0 MOV 34 N7:152 EOR
%   F8:0  "CALCULATING WEEK OF YEAR" %
%   N7:152  "ISO WEEK OF YEAR" %
% Rung: 62 %
SOR GRT F8:0 34.0 LEQ F8:0 35.0 MOV 35 N7:152 EOR
%   F8:0  "CALCULATING WEEK OF YEAR" %
%   N7:152  "ISO WEEK OF YEAR" %
% Rung: 63 %
SOR GRT F8:0 35.0 LEQ F8:0 36.0 MOV 36 N7:152 EOR
%   F8:0  "CALCULATING WEEK OF YEAR" %
%   N7:152  "ISO WEEK OF YEAR" %
% Rung: 64 %
SOR GRT F8:0 36.0 LEQ F8:0 37.0 MOV 37 N7:152 EOR
%   F8:0  "CALCULATING WEEK OF YEAR" %
%   N7:152  "ISO WEEK OF YEAR" %
% Rung: 65 %
SOR GRT F8:0 37.0 LEQ F8:0 38.0 MOV 38 N7:152 EOR
%   F8:0  "CALCULATING WEEK OF YEAR" %
%   N7:152  "ISO WEEK OF YEAR" %
% Rung: 66 %
SOR GRT F8:0 38.0 LEQ F8:0 39.0 MOV 39 N7:152 EOR
%   F8:0  "CALCULATING WEEK OF YEAR" %
%   N7:152  "ISO WEEK OF YEAR" %

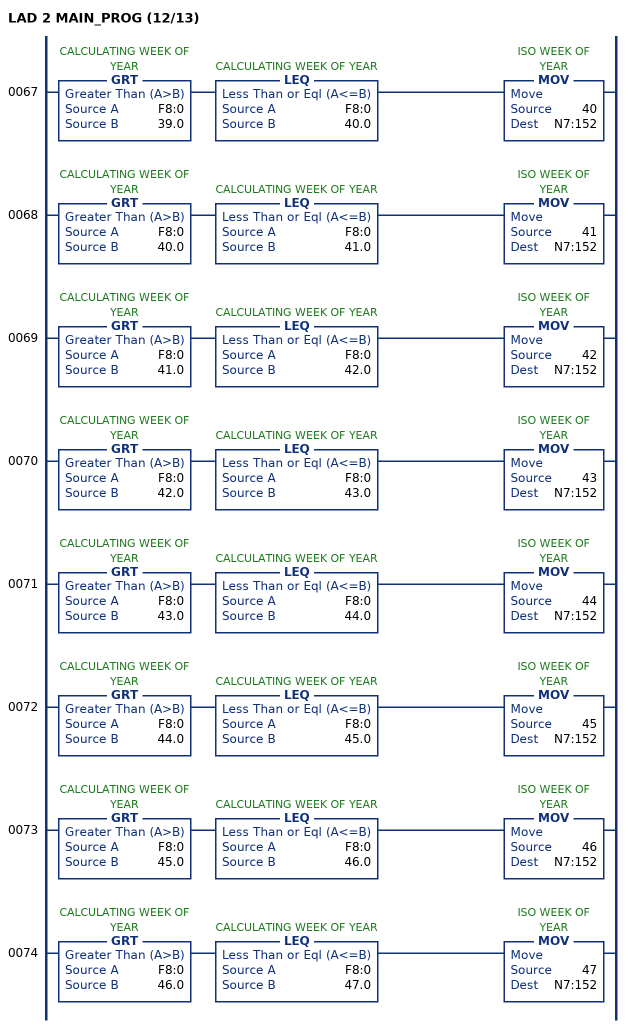
% Rung: 67 %
SOR GRT F8:0 39.0 LEQ F8:0 40.0 MOV 40 N7:152 EOR
%   F8:0  "CALCULATING WEEK OF YEAR" %
%   N7:152  "ISO WEEK OF YEAR" %
% Rung: 68 %
SOR GRT F8:0 40.0 LEQ F8:0 41.0 MOV 41 N7:152 EOR
%   F8:0  "CALCULATING WEEK OF YEAR" %
%   N7:152  "ISO WEEK OF YEAR" %
% Rung: 69 %
SOR GRT F8:0 41.0 LEQ F8:0 42.0 MOV 42 N7:152 EOR
%   F8:0  "CALCULATING WEEK OF YEAR" %
%   N7:152  "ISO WEEK OF YEAR" %
% Rung: 70 %
SOR GRT F8:0 42.0 LEQ F8:0 43.0 MOV 43 N7:152 EOR
%   F8:0  "CALCULATING WEEK OF YEAR" %
%   N7:152  "ISO WEEK OF YEAR" %
% Rung: 71 %
SOR GRT F8:0 43.0 LEQ F8:0 44.0 MOV 44 N7:152 EOR
%   F8:0  "CALCULATING WEEK OF YEAR" %
%   N7:152  "ISO WEEK OF YEAR" %
% Rung: 72 %
SOR GRT F8:0 44.0 LEQ F8:0 45.0 MOV 45 N7:152 EOR
%   F8:0  "CALCULATING WEEK OF YEAR" %
%   N7:152  "ISO WEEK OF YEAR" %
% Rung: 73 %
SOR GRT F8:0 45.0 LEQ F8:0 46.0 MOV 46 N7:152 EOR
%   F8:0  "CALCULATING WEEK OF YEAR" %
%   N7:152  "ISO WEEK OF YEAR" %
% Rung: 74 %
SOR GRT F8:0 46.0 LEQ F8:0 47.0 MOV 47 N7:152 EOR
%   F8:0  "CALCULATING WEEK OF YEAR" %
%   N7:152  "ISO WEEK OF YEAR" %

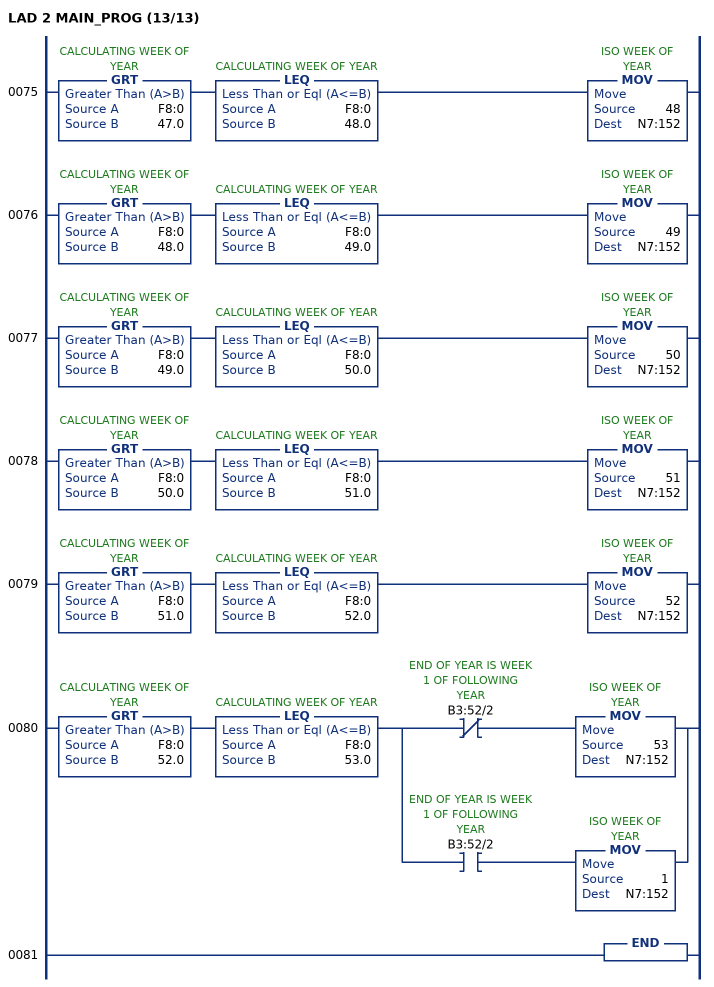
% Rung: 75 %
SOR GRT F8:0 47.0 LEQ F8:0 48.0 MOV 48 N7:152 EOR
%   F8:0  "CALCULATING WEEK OF YEAR" %
%   N7:152  "ISO WEEK OF YEAR" %
% Rung: 76 %
SOR GRT F8:0 48.0 LEQ F8:0 49.0 MOV 49 N7:152 EOR
%   F8:0  "CALCULATING WEEK OF YEAR" %
%   N7:152  "ISO WEEK OF YEAR" %
% Rung: 77 %
SOR GRT F8:0 49.0 LEQ F8:0 50.0 MOV 50 N7:152 EOR
%   F8:0  "CALCULATING WEEK OF YEAR" %
%   N7:152  "ISO WEEK OF YEAR" %
% Rung: 78 %
SOR GRT F8:0 50.0 LEQ F8:0 51.0 MOV 51 N7:152 EOR
%   F8:0  "CALCULATING WEEK OF YEAR" %
%   N7:152  "ISO WEEK OF YEAR" %
% Rung: 79 %
SOR GRT F8:0 51.0 LEQ F8:0 52.0 MOV 52 N7:152 EOR
%   F8:0  "CALCULATING WEEK OF YEAR" %
%   N7:152  "ISO WEEK OF YEAR" %
% Rung: 80 %
SOR GRT F8:0 52.0 LEQ F8:0 53.0 BST XIO B3:52/2 MOV 53 N7:152 NXB XIC B3:52/2 MOV 1 N7:152 BND EOR
%   F8:0  "CALCULATING WEEK OF YEAR" %
%   B3:52/2  "END OF YEAR IS WEEK 1 OF FOLLOWING YEAR" %
%   N7:152  "ISO WEEK OF YEAR" %
% Rung: 81 %
SOR END EOR

OTHER DOCUMENTED ADDRESSES
  N7:140  "DEGUG YEAR CHANGE TO RTC:0.YR FOR PRODUCTION"
  N7:141  "DEGUG MONTH CHANGE TO RTC:0.MON FOR PRODUCTION"
  N7:142  "DEGUG DAY CHANGE TO RTC:0.DAY FOR PRODUCTION"

DATA TABLE (non-zero values as saved)
DATA B3
% B3:50 % 0X0000 0X0000 0X0004
DATA N7
% N7:140 % 2021 1 4 0 0 0 0 0 0 0
% N7:150 % 101 0 15 0 0 0 0 0 0 0
% N7:160 % 102 1 0 0 0 0 0 0 0 0
% N7:170 % 1 2 -3 -2 -1 0 2 3 -3 -2
DATA F8
% F8:0 % 14.57143
